PROGRAM Combined_Vertical_Sample
VAR
END_VAR

astAxes[AXIS_COMBINED_VERTICAL_SAMPLE].stControl.bEnable := TRUE;
astAxes[AXIS_COMBINED_VERTICAL_SAMPLE].stInputs.bLimitBwd := astAxes[AXIS_COMBINED_VERTICAL].stInputs.bLimitBwd;
astAxes[AXIS_COMBINED_VERTICAL_SAMPLE].stInputs.bLimitFwd := astAxes[AXIS_COMBINED_VERTICAL].stInputs.bLimitFwd;

END_PROGRAM

(* stored: Version 1.1.0.1, ProductVersion 3.1.4024.11
   POU Combined_Vertical_Sample: Id {40e8365a-5831-41f5-9af5-015951ac1f91}, SpecialFunc None *)
